(* LS Electric XG5000 project: GS30_EIP_FB *)
(* GS30 EtherNet/IP function block program *)
(* PLC LSPLC *)
(* module base 0 slot 0: Input/Output Module:XEM-DN/DP32HP (DC 24V Input, Transistor Output, 32 Contacts) *)
(* module base 0 slot 1: Internal Positioning:XBF-PO06E (Open Collector Type, 6 Axis) *)
(* module base 0 slot 2: EtherNet/IP:XBL-EIPT (EtherNet/IP communication module, electrical) *)
VAR_GLOBAL
    GS30_Input00 : ARRAY[0..15] OF WORD; (* Input data to ethernet/IP GS30 drive *)
    GS30_Output00 : ARRAY[0..2] OF WORD; (* Output data to ethernet/IP GS30 drive *)
END_VAR

(* Comments on direct variables
%IX0.0.0	this is comment 1
*)

TYPE GS30_EIP_StatusAndControl_UDT : (* this is a user data type for the GS20_Drive_FB *)
STRUCT
    Direction_Command_REV : BOOL; (* FALSE =  FORWARD Direction;  TRUE =  REVERSE direction *)
    Enable_bit_function_6_11 : BOOL; (* Enables the Nth Accel/Decel and Nth Step Speed Freq functions. *)
    External_Fault_Trigger : BOOL; (* trigger an external fault mode. *)
    External_Interruption : BOOL; (* trigger an external interruption *)
    Reset_Command : BOOL; (* drive reset command *)
    Run : BOOL; (* Run drive command *)
    Stop : BOOL; (* Stop drive command *)
    Enable_JOG : BOOL; (* Jog drive. *)
    Frequency_Command : REAL; (* xx.xx Hx drive frequency command. *)
    Nth_Accel_Decel : SINT; (* Nth accel/decel functionality of drive *)
    Nth_Step_Speed_Frequency : SINT; (* Nth step speed frequency functionality of drive. *)
    Status_Actual_Motor_Speed : INT; (* xxxx RPM motor speed *)
    Status_Command_from_Comm_Keypad : BOOL; (* there is a command entered on the keypad *)
    Status_DC_Bus_Voltage : REAL; (* DC bus value *)
    Status_Decel_During_Stop : BOOL; (* 1= drive is decelerating during stop *)
    Status_Digital_Input_Counter_Value : DINT; (* Digital Input counter from drive *)
    Status_Drive_Running : BOOL; (* 1 = drive in RUN mode *)
    Status_Drive_Stopped : BOOL; (* 1 = drive is stopped *)
    Status_Freq_from_Analog_Discrete : BOOL; (* 1 = frequency is coming from an analog device input *)
    Status_Freq_from_Comm : BOOL; (* 1 = frequency is from Ethernet/IP communication *)
    Status_FreqCommand_PIDSetpoint : REAL; (* 1 = frequency is from PID setpoint *)
    Status_FWD : BOOL; (* 1 = drive is running in FWD direction *)
    Status_JOG_Active : BOOL; (* 1 = drive is in JOG mode *)
    Status_MultiSpeed_PIDStepNumber : INT; (* multispeed PID step number info *)
    Status_Output_Current : REAL; (* output current value *)
    Status_Output_Frequency : REAL; (* xx.xx Hz current frequency *)
    Status_Output_Torque : REAL; (* current torque *)
    Status_Output_Voltage : REAL; (* current output voltage *)
    Status_Parameters_Locked : BOOL; (* 1 =  paramters are locked on the drive *)
    Status_Power_Factor_Angle : REAL; (* xxx.x degrees *)
    Status_Power_Output : REAL; (* x.xxx kW *)
    Status_REV : BOOL; (* status drive is reverse movement *)
    Status_Run : BOOL; (* status of drive run *)
    Status_Standby : BOOL; (* status of drive standby mode *)
    Status_Stop : BOOL; (* status of drive stop mode *)
    Status_Transition_FWD_to_REV : BOOL; (* 1 = drive is transitioning from FWD to REV *)
    Status_Transition_REV_to_FWD : BOOL; (* 1 = drive is transitioning from REV to FWD *)
    Status_Warning_Fault_Code : INT; (* drive fault code *)
END_STRUCT;
END_TYPE

FUNCTION_BLOCK GS30_Drive_EIP_FB
(* This function block is used to control and receive status of a GS30 inverter drive. *)
VAR_INPUT
    Enable : BOOL; (* Enable the GS30 function block. *)
    InputData : ARRAY[0..15] OF WORD; (* Ethernet/IP input data array from GS30 drive *)
END_VAR
VAR_IN_OUT
    OutputData : ARRAY[0..2] OF WORD; (* Ethernet/IP output data array from GS30 drive *)
    GS30_User_UDT : GS30_EIP_StatusAndControl_UDT; (* User data type for GS30 *)
END_VAR
VAR_OUTPUT
    Active : BOOL; (* Status that GS30 function block is enabled. *)
END_VAR
VAR
    BTempOutput : ARRAY[0..5] OF BYTE; (* temporary byte array *)
    byteCount : INT; (* array counting variable *)
    byteCount2 : INT; (* array counting variable *)
    DTemp : DINT; (* temporary dint value. *)
    i : INT; (* array variable *)
    ITemp : INT; (* temporary int value *)
    Temporary_BYTE2 : BYTE; (* temporary byte storage *)
    Temporary_BYTE3 : BYTE; (* temporary byte storage. *)
    Temporary_Word : WORD; (* temporary word storage *)
    WTemp : ARRAY[0..15] OF WORD; (* temporary word array *)
    WTempOutput : ARRAY[0..2] OF WORD; (* temporary word array for output data *)
END_VAR
(***************************************************************************************************
(* 
AutomationDirect.com has provided this code for convenience. This sample code is provided "as-is" with no expressed or implied warranty. 
 If the end user includes any of the sample code (in whole or part), it is the user's responsibility to completely modify, integrate, and test any code to ensure it meets all system and 
 safety requirements for the intended application or system.
 


	The 'GS30_Drive_EIP_FB' function block uses data type WORD for the WTemp and OutputData.
		
		
									Data type:: WORD
									Input Size: 16 WORDS
									Output Size: 3 WORDS
									EDS FIle: GS30A_CM_EIP1_Rev1_0.eds -> Card with 1 Ethernet Port
									EDS File: GS30A_CM_EIP2_Rev1_0.eds -> Card with 2 Ethernet Ports
									
	***************************************************************************************************)
	
IF (Enable = TRUE) THEN		
	Active := TRUE;	
	
	(***********************
  	Mapping Input Data 
  	***********************)
 	
 	(* Copy input data to a local array *)
	FOR i:=0 TO 15 BY 1 DO
		WTemp[i] := InputData[i];
	END_FOR;
  	
  	
  	
	GS30_User_UDT.Status_Warning_Fault_Code :=  WORD_TO_INT(IN:=WTemp[0]);
	
	//Map Stop/Standby/Run.  Input Word 1, Bits 0-1
	ITemp := 0;
	ITemp.0 :=  WTemp[1].0;
	ITemp.1 := WTemp[1].1; 
	
	IF (ITemp = 0) THEN
		GS30_User_UDT.Status_Stop := TRUE;
		GS30_User_UDT.Status_Decel_During_Stop := FALSE;
		GS30_User_UDT.Status_Standby := FALSE;
		GS30_User_UDT.Status_Run := FALSE;
		
	ELSIF (ITemp = 1) THEN
		GS30_User_UDT.Status_Stop := FALSE;
		GS30_User_UDT.Status_Decel_During_Stop := TRUE;
		GS30_User_UDT.Status_Standby := FALSE;
		GS30_User_UDT.Status_Run := FALSE;	
		
	ELSIF (ITemp = 2) THEN
		GS30_User_UDT.Status_Stop := FALSE;
		GS30_User_UDT.Status_Decel_During_Stop := FALSE;
		GS30_User_UDT.Status_Standby := TRUE;
		GS30_User_UDT.Status_Run := FALSE;
	
	ELSIF (ITemp = 3) THEN	
		GS30_User_UDT.Status_Stop := FALSE;
		GS30_User_UDT.Status_Decel_During_Stop := FALSE;
		GS30_User_UDT.Status_Standby := FALSE;
		GS30_User_UDT.Status_Run := TRUE;
		
	END_IF;	
	
	//Map JOG Active Status Input Word 1, Bit 2
	GS30_User_UDT.Status_JOG_Active := WTemp[1].2;
	
	//Map Forward/Reverse Status.  Input Word 1, Bits 3-4
	ITemp := 0;
	ITemp.0 :=  WTemp[1].3;
	ITemp.1 := WTemp[1].4; 
	
	IF (ITemp = 0) THEN
		GS30_User_UDT.Status_FWD := TRUE;
		GS30_User_UDT.Status_Transition_REV_to_FWD := FALSE;
		GS30_User_UDT.Status_Transition_FWD_to_REV := FALSE;
		GS30_User_UDT.Status_REV := FALSE;
		
	ELSIF (ITemp = 1) THEN
		GS30_User_UDT.Status_FWD := FALSE;
		GS30_User_UDT.Status_Transition_REV_to_FWD := TRUE;
		GS30_User_UDT.Status_Transition_FWD_to_REV := FALSE;
		GS30_User_UDT.Status_REV := FALSE;	
		
	ELSIF (ITemp = 2) THEN
		GS30_User_UDT.Status_FWD := FALSE;
		GS30_User_UDT.Status_Transition_REV_to_FWD := FALSE;
		GS30_User_UDT.Status_Transition_FWD_to_REV := TRUE;
		GS30_User_UDT.Status_REV := FALSE;
	
	ELSIF (ITemp = 3) THEN	
		GS30_User_UDT.Status_FWD := TRUE;
		GS30_User_UDT.Status_Transition_REV_to_FWD := FALSE;
		GS30_User_UDT.Status_Transition_FWD_to_REV := FALSE;
		GS30_User_UDT.Status_REV := TRUE;
		
	END_IF;	
	
	//Map Freq from Comm status.   Input Word 1, Bit 8
	GS30_User_UDT.Status_Freq_from_Comm := WTemp[1].8;
	
	//Map Freq from Analog/Discrete.   Input Word 1, Bit 9
	GS30_User_UDT.Status_Freq_from_Analog_Discrete := WTemp[1].9;
	
	//Map Command from Comm/Keypad.  Input Word 1, Bit 10
	GS30_User_UDT.Status_Command_from_Comm_Keypad := WTemp[1].10;
	
	//Map Parameters locked status.  Input Word 1, Bit 11
	GS30_User_UDT.Status_Parameters_Locked := WTemp[1].11;
	
	//Map Running Status.  Input Word 1, Bit 12
	GS30_User_UDT.Status_Drive_Running :=  WTemp[1].12;
	GS30_User_UDT.Status_Drive_Stopped := NOT(WTemp[1].12);
	
	//Map Frequency Commanded / PID Setpoint.   Input Word 2.   6000 = 60.00 Hz.  Convert WORD to REAL value.
	DTemp := WORD_TO_DINT(IN:=WTemp[2]);
	GS30_User_UDT.Status_FreqCommand_PIDSetpoint := DINT_TO_REAL(IN:=DTemp) / 100.00;
	
	//Map Output Frequency.   Input Word 3.    6000 = 60.00 Hz.  Convert WORD to REAL value.
	DTemp := WORD_TO_DINT(IN:=WTemp[3]);
	GS30_User_UDT.Status_Output_Frequency := DINT_TO_REAL(IN:=DTemp) / 100.00;
	
	//Map Output Current.   Input Word 4.    6000 = 60.00 A.   Convert WORD to REAL value.
	DTemp := WORD_TO_DINT(IN:=WTemp[4]);
	GS30_User_UDT.Status_Output_Current := DINT_TO_REAL(IN:=DTemp) / 100.00;
	
	//Map DC Bus Voltage.   Input Word 5.    6000 = 600.0 Vdc.  Convert WORD to REAL value.
	DTemp := WORD_TO_DINT(IN:=WTemp[5]);
	GS30_User_UDT.Status_DC_Bus_Voltage := DINT_TO_REAL(IN:=DTemp) / 10.00;
	
	//Map Output Voltage.   Input Word 6.    6000 = 600.0 VAC.  Convert WORD to REAL value.
	DTemp := WORD_TO_DINT(IN:=WTemp[6]);
	GS30_User_UDT.Status_Output_Voltage := DINT_TO_REAL(IN:=DTemp) / 10.00;
	
	//Map Multi-Speed / PID Step Number.   Input Word 7.   Convert WORD to INT value.
	GS30_User_UDT.Status_MultiSpeed_PIDStepNumber := WORD_TO_INT(IN:=WTemp[7]);
	
	//Map Digital Input Counter Value.   Input Word 9.   Convert WORD to DINT value.
	GS30_User_UDT.Status_Digital_Input_Counter_Value := WORD_TO_DINT(IN:=WTemp[9]);
	
	//Map Power Factor Angle .   Input Word 10.    6000 = 600.0 degrees.  Convert WORD to REAL value.
	DTemp := WORD_TO_DINT(IN:=WTemp[10]);
	GS30_User_UDT.Status_Power_Factor_Angle := DINT_TO_REAL(IN:=DTemp) / 10.00;
	
	//Map Output Torque .   Input Word 11.    6000 = 600.0 %.  Convert WORD to REAL value.
	DTemp := WORD_TO_DINT(IN:=WTemp[11]);
	GS30_User_UDT.Status_Output_Torque := DINT_TO_REAL(IN:=DTemp) / 10.00;
	
	//Map actual motor speed (RPM) .   Input Word 12.    XXXX RPM.  Convert WORD to INT value.
	GS30_User_UDT.Status_Actual_Motor_Speed := WORD_TO_INT(IN:=WTemp[12]);
	
	//Map power output .   Input Word 15.    XXXX = X.xxx kW.  Convert WORD to REAL value.
	DTemp := WORD_TO_DINT(IN:=WTemp[15]);
	GS30_User_UDT.Status_Power_Output := DINT_TO_REAL(IN:=DTemp) / 1000.00;
	
	
	(***********************
  	Mapping Output Data 
  	***********************)
 	
 	//Map Run/Stop/JOG Command.  Output Word 0, Bits 0-1.     0= No Function; 1=STOP; 2= RUN; 3=Enable JOG
  	ITemp := 0;
  	
  	IF (GS30_User_UDT.Stop = TRUE) THEN
  		ITemp := 1;
  		
  	ELSIF	(GS30_User_UDT.Enable_JOG = TRUE) AND (GS30_User_UDT.Stop = FALSE) THEN
  		ITemp := 3;
  		
  	ELSIF  (GS30_User_UDT.Run = TRUE) AND (GS30_User_UDT.Stop = FALSE) THEN
  		ITemp := 2;
  	
  	END_IF;	
  	
  	WTempOutput[0].0 := ITemp.0;
  	WTempOutput[0].1 := ITemp.1;
  	
  	
  	//Map forward/reverse command.   Output Word 0, Bits 4-5.     0= No Function; 1 = Forward Command; 2 = Reverse Command; 3 = No Function.
  	IF (GS30_User_UDT.Direction_Command_REV = TRUE) THEN
  		WTempOutput[0].4 := 0;
  		WTempOutput[0].5 := 1;
  	ELSE
  		WTempOutput[0].4 := 1;
  		WTempOutput[0].5 := 0;		
  	END_IF;
  	
  	
  	//Map Nth Accel/Decel.  Output Word 0, Bits 6-7.  0 = 1st Accel/Decel; 1 = 2nd Accel/Decel; 2 = 3rd Accel/Decel;  3 = 4th Accel/Decel
  	WTempOutput[0].6 := GS30_User_UDT.Nth_Accel_Decel.0;
  	WTempOutput[0].7 := GS30_User_UDT.Nth_Accel_Decel.1;
  	
  	(* Map Nth Step Speed Frequency.   Output Word 0, Bits 8-11.  0
   			0 = Master Speed; 1 = 1st Step Speed Frequency; 2 = 2nd Step Speed Frequency;  3 = 3rd Step Speed Frequency; 4 = 4th Step Speed Frequency
   			5 = 5th Step Speed Frequency, 6 = 6th Step Speed Frequency,  7= 7th Step Speed Frequency,  8 = 8th Step Speed Frequency, 9 = 9th Step Speed Frequency,
   			10 = 10th Step Speed Frequency, 11 = 11th Step Speed Frequency,  12 = 12th Step Speed Frequency, 13 = 13th Step Speed Frequency, 14 = 14th Step Speed Frequency
   			15 = 15th Step Speed Frequency.
   		*)	
  	WTempOutput[0].8 := GS30_User_UDT.Nth_Step_Speed_Frequency.0;
  	WTempOutput[0].9 := GS30_User_UDT.Nth_Step_Speed_Frequency.1;
  	WTempOutput[0].10 := GS30_User_UDT.Nth_Step_Speed_Frequency.2;
  	WTempOutput[0].11 := GS30_User_UDT.Nth_Step_Speed_Frequency.3;
  	
  	//Map Enable bit function 6-11.  Output Word 0, Bit 12.   Enables the Nth Accel/Decel and Nth Step Speed Frequency function.
  	WTempOutput[0].12 := GS30_User_UDT.Enable_bit_function_6_11;
 	
 	//Map Frequency Command.  Output Word 1.   Convert Real to INT.  60.00 Hz = 6000
 	DTemp := REAL_TO_DINT(IN:=GS30_User_UDT.Frequency_Command * 100.0);
 	WTempOutput[1] := DINT_TO_WORD(DTemp);
 	
 	//Map External Fault Trigger.  Output Word 2, Bit 0
 	WTempOutput[2].0 := GS30_User_UDT.External_Fault_Trigger;
 	
  	//Map Reset Command.  Output Word 2, Bit 1
 	WTempOutput[2].1 := GS30_User_UDT.Reset_Command;
 	
  	//Map External Interrupt.   Output Word 2, Bit 2
 	WTempOutput[2].2 := GS30_User_UDT.External_Interruption;
 	
 		

 	
 	OutputData := ARY_MOVE(MOVE_NUM:=3, IN:=WTempOutput, IN_INDX:=0, OUT_INDX:=0);


ELSE
	Active := FALSE;
END_IF;
END_FUNCTION_BLOCK

PROGRAM FB_Usage_LD (* task: Scan Program *)
VAR
    fbActive : BOOL;
    GS30_INST00 : GS30_Drive_EIP_FB; (* GS30 Control function block *)
    GS30_User_UDT : GS30_EIP_StatusAndControl_UDT; (* User data type for GS30 control *)
END_VAR
VAR_EXTERNAL
    GS30_Input00 : ARRAY[0..15] OF WORD; (* Input data to ethernet/IP GS30 drive *)
    GS30_Output00 : ARRAY[0..2] OF WORD; (* Output data to ethernet/IP GS30 drive *)
END_VAR

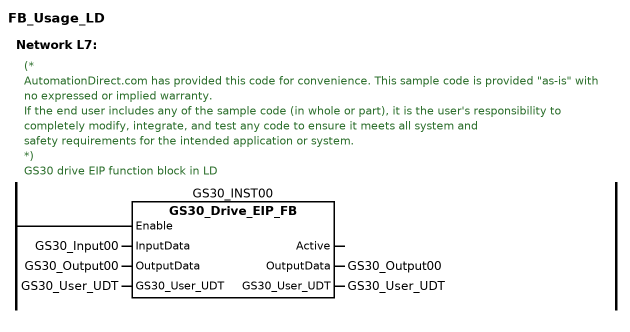
(* ( * / AutomationDirect.com has provided this code for convenience. This sample code is provided "as-is" with no expressed or implied warranty. / If the end user includes any of the sample code (in whole or part), it is the user's responsibility to completely modify, integrate, and test any code to ensure it meets all system and / safety requirements for the intended application or system. / * ) *)
(* GS30 drive EIP function block in LD *)
(* Rung L7 *)
GS30_INST00(Enable := TRUE, InputData := GS30_Input00, OutputData := GS30_Output00, GS30_User_UDT := GS30_User_UDT, OutputData => GS30_Output00, GS30_User_UDT => GS30_User_UDT);
END_PROGRAM

PROGRAM FB_Usage_ST (* task: Scan Program *)
(*  *)
VAR
    Enable : BOOL;
    fbActive : BOOL;
    GS30_Inst00 : GS30_Drive_EIP_FB; (* GS30 function block *)
    GS30_User_UDT : GS30_EIP_StatusAndControl_UDT; (* User data type for GS30 control *)
    ITemp : INT;
END_VAR
VAR_EXTERNAL
    GS30_Input00 : ARRAY[0..15] OF WORD; (* Input data to ethernet/IP GS30 drive *)
    GS30_Output00 : ARRAY[0..2] OF WORD; (* Output data to ethernet/IP GS30 drive *)
END_VAR
(* 
AutomationDirect.com has provided this code for convenience. This sample code is provided "as-is" with no expressed or implied warranty. 
 If the end user includes any of the sample code (in whole or part), it is the user's responsibility to completely modify, integrate, and test any code to ensure it meets all system and 
 safety requirements for the intended application or system.
 *)

Enable := TRUE;


//GS30_Inst00(Enable:=TRUE, InputData:=GS30_Input00, OutputData:=GS30_Output00, GS30_User_UDT:=GS30_User_UDT, Active=>fbActive);
END_PROGRAM